Staubli VAL3: changeValue.pgx

public program changeValue(num& x_nValue[] (dimensions=1), num x_nMin (dimensions=1), num x_nMax (dimensions=1), num x_nX (dimensions=1), num x_nY (dimensions=1), string& x_sItems[] (dimensions=1))
  local num l_nOldValue[2]
  local string l_sItem
  local string l_sMessage
  local bool l_bComma
  local string l_sEmpty
begin
  //---------------------------------
  // Staubli copyright 2005
  //                By toneage
  //[Public]-------------------------
  //
  // x_nValue:  num to change
  // x_nMax:    max value
  // x_nMin:    min value
  // x_nX:      X position
  // x_nY:      Y position
  // x_sItems   message
  //
  // look if the value is between max and min
  //
  if x_nMin>x_nMax
    return
  endIf
  //
  // print the line in white
  //
  // call listCleanLine()
  //
  call nullKey(nKey)
  l_nOldValue[1]=round(x_nValue)
  x_nValue=(round(x_nValue*1000))/1000
  l_nOldValue=x_nValue
  // check if is using the comma or not
  if l_nOldValue!=l_nOldValue[1]
    l_bComma=true
  else
    l_bComma=false
  endIf
  // start
  call clear(0,13)
  do
    if x_sItems==""
      //
      //  use the get num
      //
      if l_bComma
        call strfill(l_sEmpty,len(toString(".3",x_nValue)),l_sEmpty)
      else
        call strfill(l_sEmpty,len(toString(".3",x_nValue)),l_sEmpty)
      endIf
      call type(x_nX,x_nY,l_sEmpty)
      gotoxy(x_nX,x_nY)
      nKey=get(x_nValue)
      // check the comma again
      if round(x_nValue)!=x_nValue
        l_bComma=true
      endIf
      //
      // CHECK for MIN MAX VALUE
      //
      if x_nMax!=x_nMin or x_nMin!=0
        if x_nValue>x_nMax
          //
          // ask if you want to continue
          //
          popUpMsg("MAX: "+toString(".2",x_nMax))
          x_nValue=l_nOldValue
          //x_nValue=x_nMax
          nKey=-1
        else
          if x_nValue<x_nMin
            //
            popUpMsg("MIN: "+toString(".2",x_nMin))
            //x_nValue=x_nMin
            x_nValue=l_nOldValue
            nKey=-1
          endIf
        endIf
      endIf
      //
      // UPDATE THE VALUE
      //
      if l_bComma
        call type(x_nX,x_nY,toString(".2",x_nValue))
      else
        call type(x_nX,x_nY,toString("",x_nValue))
      endIf
    else
      // STRING CHOICE
      nKey=getKey()
      switch nKey
        // CHANGE THE ITEMS ARRAY
        case 261
          // UP
          x_nValue=abs((x_nValue+1)%size(x_sItems))
        break
        case 266
          // DOWN
          x_nValue=abs((x_nValue+size(x_sItems)-1)%size(x_sItems))
        break
      endSwitch
      //
      // UPDATE THE VALUE
      //
      setTextMode(3)
      call typeLen(x_nX,x_nY,x_sItems[x_nValue],8)
      setTextMode(0)
    endIf
    // release the resource
    delay(0)
  until nKey==270 or nKey==255
  if nKey==255
    bUseEscape=true
    x_nValue=l_nOldValue
    if x_sItems!=""
      x_sItems=x_sItems[l_nOldValue]
    endIf
  else
    bUseEscape=false
  endIf
  // leave the resource
  delay(0)
end
